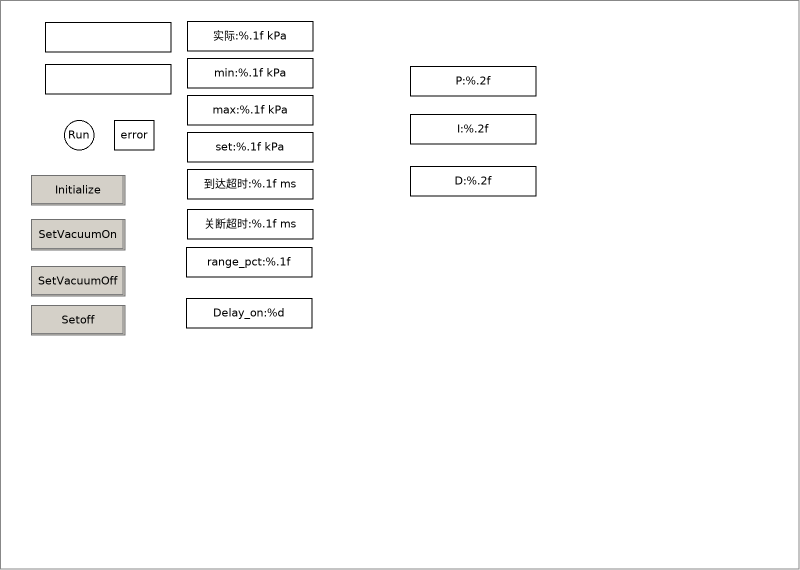
VISUALIZATION VIS_TabVac  // 800x570
    Rectangle (45,22 126x30), text list: 'TextList_tabvac_state', text index: GVL_API.stTableVacuum[1].state
    Button (31,175 94x30), "Initialize", colour toggle: GVL_API.stTableVacuum[1].Initialize
        toggle GVL_API.stTableVacuum[1].Initialize
    Button (31,219 94x31), "SetVacuumOn", colour toggle: GVL_API.stTableVacuum[1].SetVacuumOn
        toggle GVL_API.stTableVacuum[1].SetVacuumOn
        OnMouseDown: execute { GVL_API.stAxis[1].homingvelocity:=100; }
    Button (31,266 94x30), "SetVacuumOff", colour toggle: GVL_API.stTableVacuum[1].SetVacuumOff
        toggle GVL_API.stTableVacuum[1].SetVacuumOff
    Button (31,305 94x30), "Setoff", colour toggle: GVL_API.stTableVacuum[1].Setoff
        toggle GVL_API.stTableVacuum[1].Setoff
    Rectangle (187,21 126x30), "实际:%.1f kPa", text variable: GVL_API.stTableVacuum[1].vacuum_measured
        OnMouseDown: write GVL_API.stTableVacuum[1].vacuum_measured via Default
    Rectangle (187,58 126x30), "min:%.1f kPa", text variable: GVL_API.stTableVacuum[1].vacuum_min
        OnMouseDown: write GVL_API.stTableVacuum[1].vacuum_min via Default
    Rectangle (187,95 126x30), "max:%.1f kPa", text variable: GVL_API.stTableVacuum[1].vacuum_max
        OnMouseDown: write GVL_API.stTableVacuum[1].vacuum_max via Default
    Rectangle (187,169 126x30), "到达超时:%.1f ms", text variable: GVL_API.stTableVacuum[1].vacuum_timeout
        OnMouseDown: write GVL_API.stTableVacuum[1].vacuum_timeout via Default
    Rectangle (187,209 126x30), "关断超时:%.1f ms", text variable: GVL_API.stTableVacuum[1].vacuum_off_timeout
        OnMouseDown: write GVL_API.stTableVacuum[1].vacuum_off_timeout via Default
    Ellipse (64,120 30x30), "Run", colour toggle: stOutput.bqVacRun[1]
    Rectangle (187,132 126x30), "set:%.1f kPa", text variable: GVL_API.stTableVacuum[1].setpoint
        OnMouseDown: write GVL_API.stTableVacuum[1].setpoint via Default
    Rectangle (186,247 126x30), "range_pct:%.1f", text variable: GVL_API.stTableVacuum[1].setpoint_range_pct
        OnMouseDown: write GVL_API.stTableVacuum[1].setpoint_range_pct via Default
    Rectangle (45,64 126x30), text list: 'TextList_tabvac_errorid', text index: GVL_API.stTableVacuum[1].error_code
    Rectangle (410,66 126x30), "P:%.2f", text variable: GVL_API.stTableVacuum[1].ctrlP
        OnMouseDown: write GVL_API.stTableVacuum[1].ctrlP via Default
    Rectangle (410,114 126x30), "I:%.2f", text variable: GVL_API.stTableVacuum[1].ctrlI
        OnMouseDown: write GVL_API.stTableVacuum[1].ctrlI via Default
    Rectangle (410,166 126x30), "D:%.2f", text variable: GVL_API.stTableVacuum[1].ctrlD
        OnMouseDown: write GVL_API.stTableVacuum[1].ctrlD via Default
    RoundedRectangle (114,120 40x30), "error", colour toggle: GVL_API.stTableVacuum[1].Error
    Rectangle (186,298 126x30), "Delay_on:%d", text variable: HMI_Vac_dely_on
        OnMouseDown: write HMI_Vac_dely_on via Default, min 0
END_VISUALIZATION

(* stored: Version 1.1.0.1, ProductVersion 3.1.4024.11
   Visu VIS_TabVac: Id {44aeeccc-cfae-4d30-aeaf-d870f7cd4e7a} *)
